FUNCTION_BLOCK FB_FORECAST_TIMER (* Forwards inputs and delegates request to UD every minute and to FREQ every RS minutes *)
  (* Standard: 61499-2 *)
  (* Version 0.0, 2017-05-17, Marc Jakobi, HTW Berlin *)
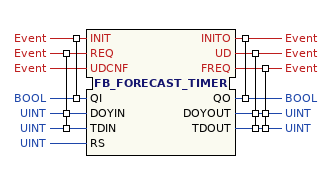
  EVENT_INPUT
    INIT WITH QI; (* Initialization Request *)
    REQ WITH TDIN, DOYIN; (* Normal Execution Request *)
    UDCNF; (* Confirmation of completed update/s *)
  END_EVENT
  EVENT_OUTPUT
    INITO WITH QO; (* Initialization Confirm *)
    UD WITH DOYOUT, TDOUT; (* Memory update request for PowerForecaster FBs *)
    FREQ WITH TDOUT, DOYOUT; (* Forecast request for PowerForecaster FBs *)
  END_EVENT
  VAR_INPUT
    QI : BOOL; (* Input event qualifier *)
    DOYIN : UINT := 1; (* Day of the year [1..365] *)
    TDIN : UINT; (* Time of day [min] [0..1439] *)
    RS : UINT := 15; (* Frequency [min] to send out FREQ event *)
  END_VAR
  VAR_OUTPUT
    QO : BOOL; (* Output event qualifier *)
    DOYOUT : UINT := 1; (* Day of the year [1..365] *)
    TDOUT : UINT := 0; (* Time of day [min] [0..1439] *)
  END_VAR
  VAR
    COUNTER : UINT := 0; (* Counts from 1 to 15 *)
    LASTTDIN : INT := -1; (* Cache for TDIN *)
  END_VAR
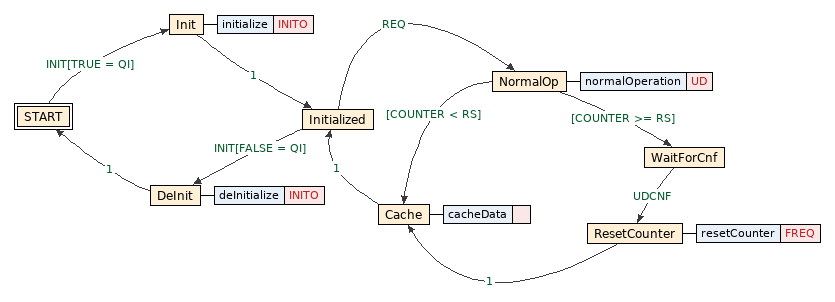
  EC_STATES
    START; (* Initial State *)
    Init : initialize -> INITO; (* Initialization *)
    NormalOp : normalOperation -> UD; (* Normal execution *)
    Initialized;
    DeInit : deInitialize -> INITO;
    ResetCounter : resetCounter -> FREQ;
    Cache : cacheData;
    WaitForCnf;
  END_STATES
  EC_TRANSITIONS
    START TO Init := INIT[TRUE = QI];
    Init TO Initialized := 1;
    Initialized TO NormalOp := REQ;
    DeInit TO START := 1;
    Initialized TO DeInit := INIT[FALSE = QI];
    NormalOp TO Cache := [COUNTER < RS];
    ResetCounter TO Cache := 1;
    Cache TO Initialized := 1;
    NormalOp TO WaitForCnf := [COUNTER >= RS];
    WaitForCnf TO ResetCounter := UDCNF;
  END_TRANSITIONS
  ALGORITHM initialize IN ST: (* Initialization algorithm *)
COUNTER := 0;
QO := QI;
  END_ALGORITHM
  ALGORITHM deInitialize IN ST: (* Normally executed algorithm *)
COUNTER := 0;
QO := FALSE;
  END_ALGORITHM
  ALGORITHM normalOperation IN ST: (* passes inputs to outputs and increments COUNTER by 1 *)
VAR
	timeSinceLastExecution : INT;
END_VAR;
/*
 * Used internal vars and inputs:
 * COUNTER, DOYIN, DOYOUT, TDIN, TDOUT : UINT;
 * LASTTDIN : INT;
 */
// Increment counter
timeSinceLastExecution := UINT_TO_INT(TDIN) - LASTTDIN;
IF timeSinceLastExecution < 0 THEN // If last minute of yesterday was skipped
	timeSinceLastExecution := timeSinceLastExecution + 1440; // add 1440 minutes to correct time
END_IF;
COUNTER := COUNTER + INT_TO_UINT(timeSinceLastExecution);
// Set outputs
TDOUT := TDIN;
DOYOUT := DOYIN;
  END_ALGORITHM
  ALGORITHM resetCounter IN ST: (* resets COUNTER *)
WHILE COUNTER >= RS DO // While loop in case for some reason minutes were skipped
	COUNTER := COUNTER - RS;
END_WHILE;
  END_ALGORITHM
  ALGORITHM cacheData IN ST: (* caches inputs for next execution *)
IF TDIN >= 1439 THEN
	LASTTDIN := -1; // Reset if end of day
ELSE
	LASTTDIN := UINT_TO_INT(TDIN); // Otherwise cache input
END_IF;
  END_ALGORITHM
END_FUNCTION_BLOCK
